{attribute 'GeneratedUsingTerminal: EK1100-0000-0018'}
{attribute addProperty BoxType "EK1100-0000-0018"}
{attribute addProperty Id "Beckhoff_ER3xxxEK1122Beckhoff_ER3xxxEK1122_4F8E32D9618"}
{attribute addProperty CRC "1487295449"}
{attribute addProperty Size "618"}
TYPE Beckhoff_ER3xxx_58A653D9 EXTENDS EK1100_1FC0878B :
STRUCT
	{attribute addProperty Name "Beckhoff ER3xxxEK1122"}
	{attribute addProperty PreviousPort "Beckhoff ER3xxx : B"}
	Beckhoff_ER3xxxEK1122 : Beckhoff_ER3xxxEK1122_4F8E32D9;
END_STRUCT
END_TYPE

(* stored: Version 1.2.0.0, ProductVersion 3.1.4024.9
   DUT Beckhoff_ER3xxx_58A653D9: Id {fc9f75dc-5da2-4793-a1ed-bf3678259bad} *)
